FUNCTION F_AddPaddingUDINT : STRING
VAR_INPUT
	nNumber:		UDINT;
	nSize:			UINT;
END_VAR
VAR
	sTemp: STRING;
END_VAR

sTemp := UDINT_TO_STRING(nNumber);

WHILE LEN(sTemp) < nSize DO
	sTemp := CONCAT('0',sTemp);
END_WHILE

F_AddPaddingUDINT := sTemp;

END_FUNCTION

(* stored: Version 1.1.0.1, ProductVersion 3.1.4024.15
   POU F_AddPaddingUDINT: Id {1cc5d340-60cc-49dc-a777-719c2cf79b73}, SpecialFunc None *)
